FUNCTION_BLOCK EMGYSTOP
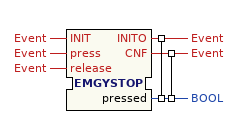
  EVENT_INPUT
    INIT;
    press;
    release;
  END_EVENT
  EVENT_OUTPUT
    INITO WITH pressed;
    CNF WITH pressed;
  END_EVENT
  VAR_OUTPUT
    pressed : BOOL;
  END_VAR
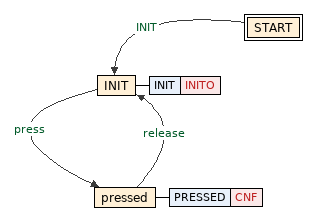
  EC_STATES
    START;
    pressed : PRESSED -> CNF;
    INIT : INIT -> INITO;
  END_STATES
  EC_TRANSITIONS
    START TO INIT := INIT;
    INIT TO pressed := press;
    pressed TO INIT := release;
  END_TRANSITIONS
  ALGORITHM INIT IN ST:
pressed := FALSE;
  END_ALGORITHM
  ALGORITHM PRESSED IN ST:
pressed := TRUE;
  END_ALGORITHM
END_FUNCTION_BLOCK
